PROGRAM Batch_Controller
  VAR_EXTERNAL
    Safety_OK : BOOL;
    Level : REAL;
    Temperature : REAL;
    Pressure : REAL;
    Weight : REAL;
    Ingredient_A_Request : BOOL;
    Ingredient_B_Request : BOOL;
    Discharge_Request : BOOL;
    Packaging_Request : BOOL;
    Mixer_Request : BOOL;
    Batch_State_Code : INT;
    Batch : ST_BATCH;
  END_VAR
  VAR
    Batch_Start : BOOL;
    Batch_Stop : BOOL;
    Batch_Reset : BOOL;
    Fill_A_Active : BOOL;
    Fill_A_Done : BOOL;
    Fill_B_Active : BOOL;
    Fill_B_Done : BOOL;
    Batch_Target : REAL;
    Mix_Active : BOOL;
    Mix_Done : BOOL;
    Mix_Timer : TON;
    Discharge_Active : BOOL;
    Discharge_Done : BOOL;
    Packaging_Active : BOOL;
    Packaging_Done : BOOL;
    Packaging_Timer : TON;
    Batch_Complete : BOOL;
    Batch_Start_Trig : R_TRIG;
  END_VAR
  VAR  (* added by the conversion: wires and edge detectors of the diagram *)
    _State_Transition12_ENO : BOOL;
    _State_Transition12_OUT : INT;
  END_VAR

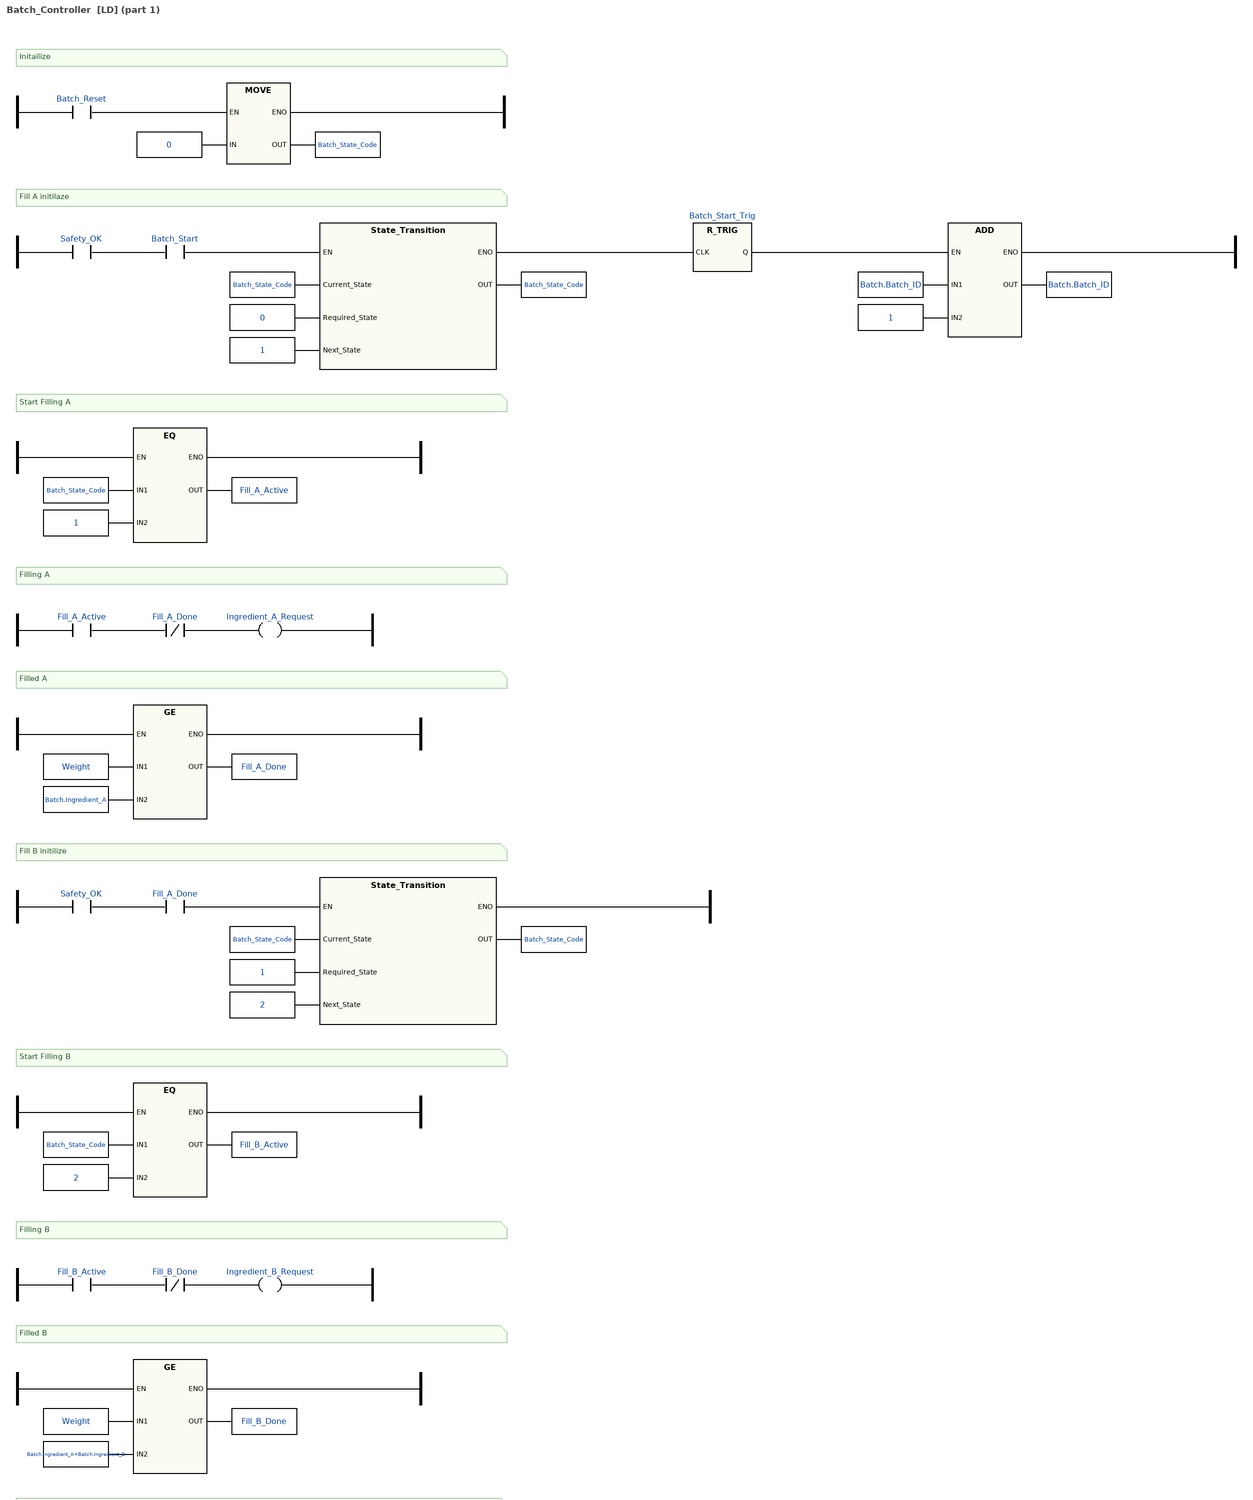
(* LD diagram, written out as Structured Text *)
(* Initailize *)
IF Batch_Reset THEN Batch_State_Code := 0; END_IF;
(* Fill A initilaze *)
_State_Transition12_OUT := State_Transition(EN := Safety_OK AND Batch_Start, Current_State := Batch_State_Code, Required_State := 0, Next_State := 1, ENO => _State_Transition12_ENO);
IF _State_Transition12_ENO THEN Batch_State_Code := _State_Transition12_OUT; END_IF;
Batch_Start_Trig(CLK := _State_Transition12_ENO);
IF Batch_Start_Trig.Q THEN Batch.Batch_ID := Batch.Batch_ID + 1; END_IF;
(* Start Filling A *)
Fill_A_Active := Batch_State_Code = 1;
(* Filling A *)
Ingredient_A_Request := Fill_A_Active AND NOT Fill_A_Done;
(* Filled A *)
Fill_A_Done := Weight >= Batch.Ingredient_A;
(* Fill B initilize *)
IF Safety_OK AND Fill_A_Done THEN Batch_State_Code := State_Transition(Batch_State_Code, 1, 2); END_IF;
(* Start Filling B *)
Fill_B_Active := Batch_State_Code = 2;
(* Filling B *)
Ingredient_B_Request := Fill_B_Active AND NOT Fill_B_Done;
(* Filled B *)
Fill_B_Done := Weight >= (Batch.Ingredient_A+Batch.Ingredient_B);
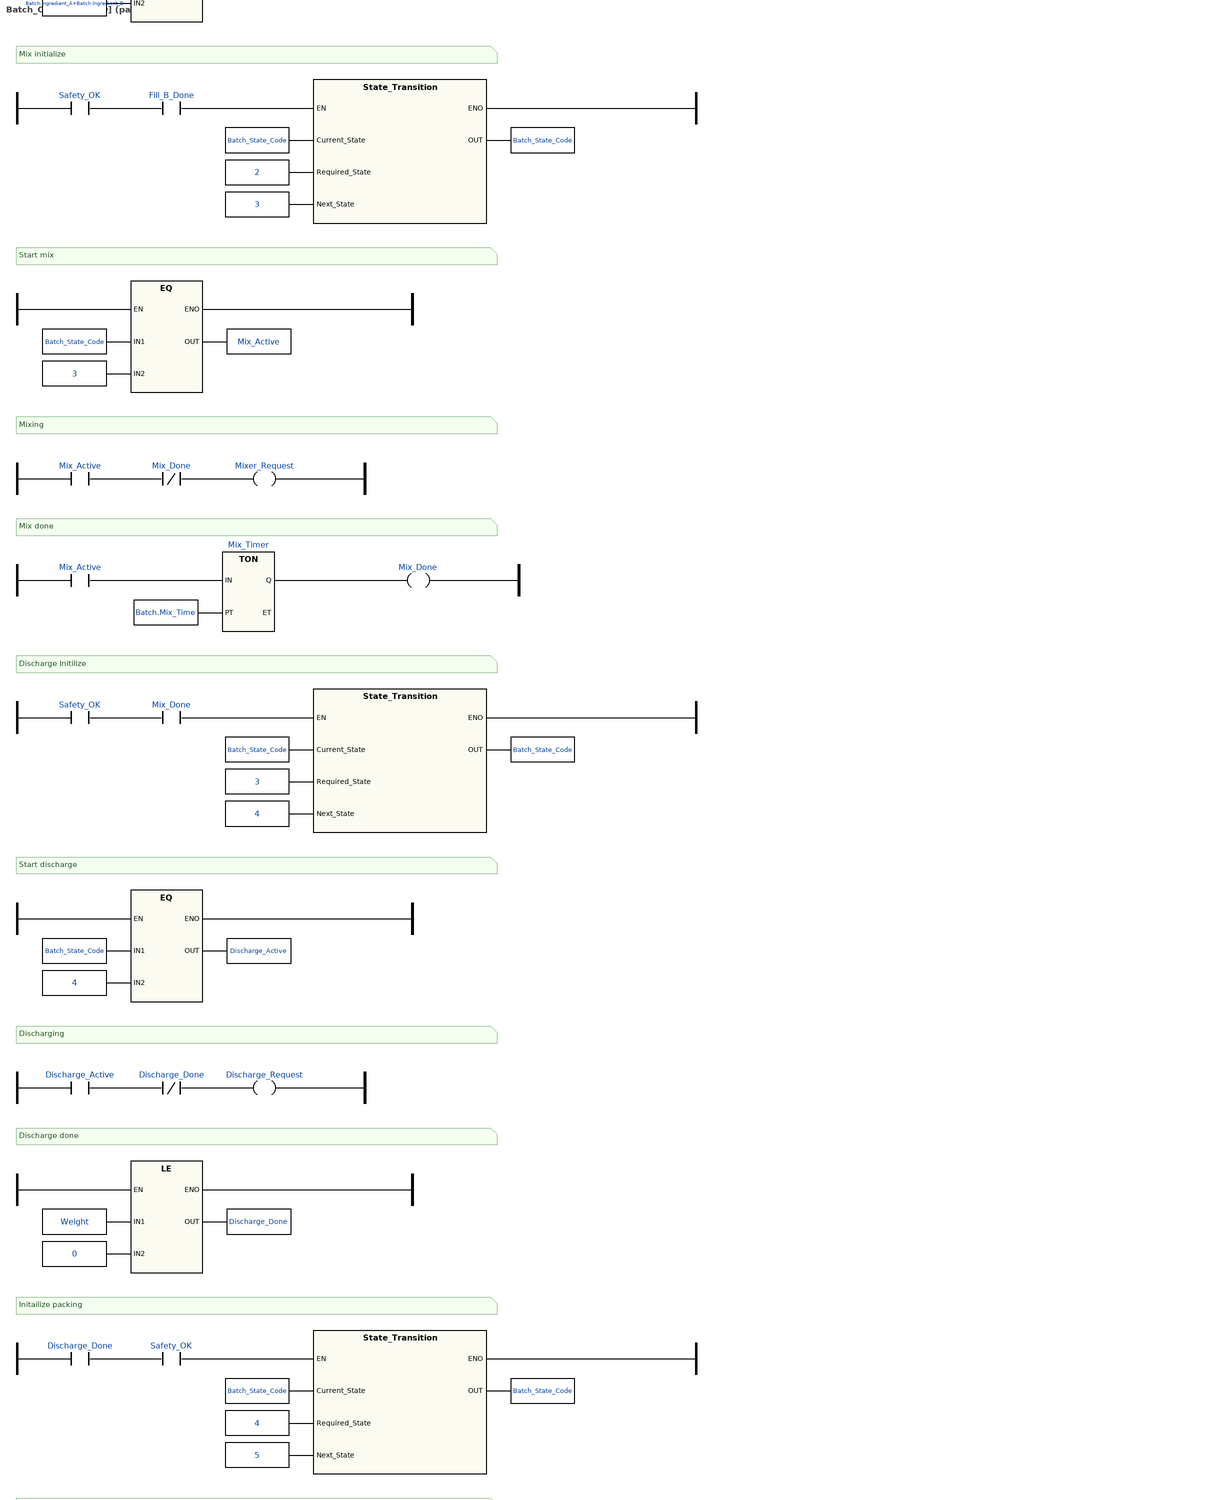
(* Mix initialize *)
IF Safety_OK AND Fill_B_Done THEN Batch_State_Code := State_Transition(Batch_State_Code, 2, 3); END_IF;
(* Start mix *)
Mix_Active := Batch_State_Code = 3;
(* Mixing *)
Mixer_Request := Mix_Active AND NOT Mix_Done;
(* Mix done *)
Mix_Timer(IN := Mix_Active, PT := Batch.Mix_Time);
Mix_Done := Mix_Timer.Q;
(* Discharge Initilize *)
IF Safety_OK AND Mix_Done THEN Batch_State_Code := State_Transition(Batch_State_Code, 3, 4); END_IF;
(* Start discharge *)
Discharge_Active := Batch_State_Code = 4;
(* Discharging *)
Discharge_Request := Discharge_Active AND NOT Discharge_Done;
(* Discharge done *)
Discharge_Done := Weight <= 0;
(* Initailize packing *)
IF Discharge_Done AND Safety_OK THEN Batch_State_Code := State_Transition(Batch_State_Code, 4, 5); END_IF;
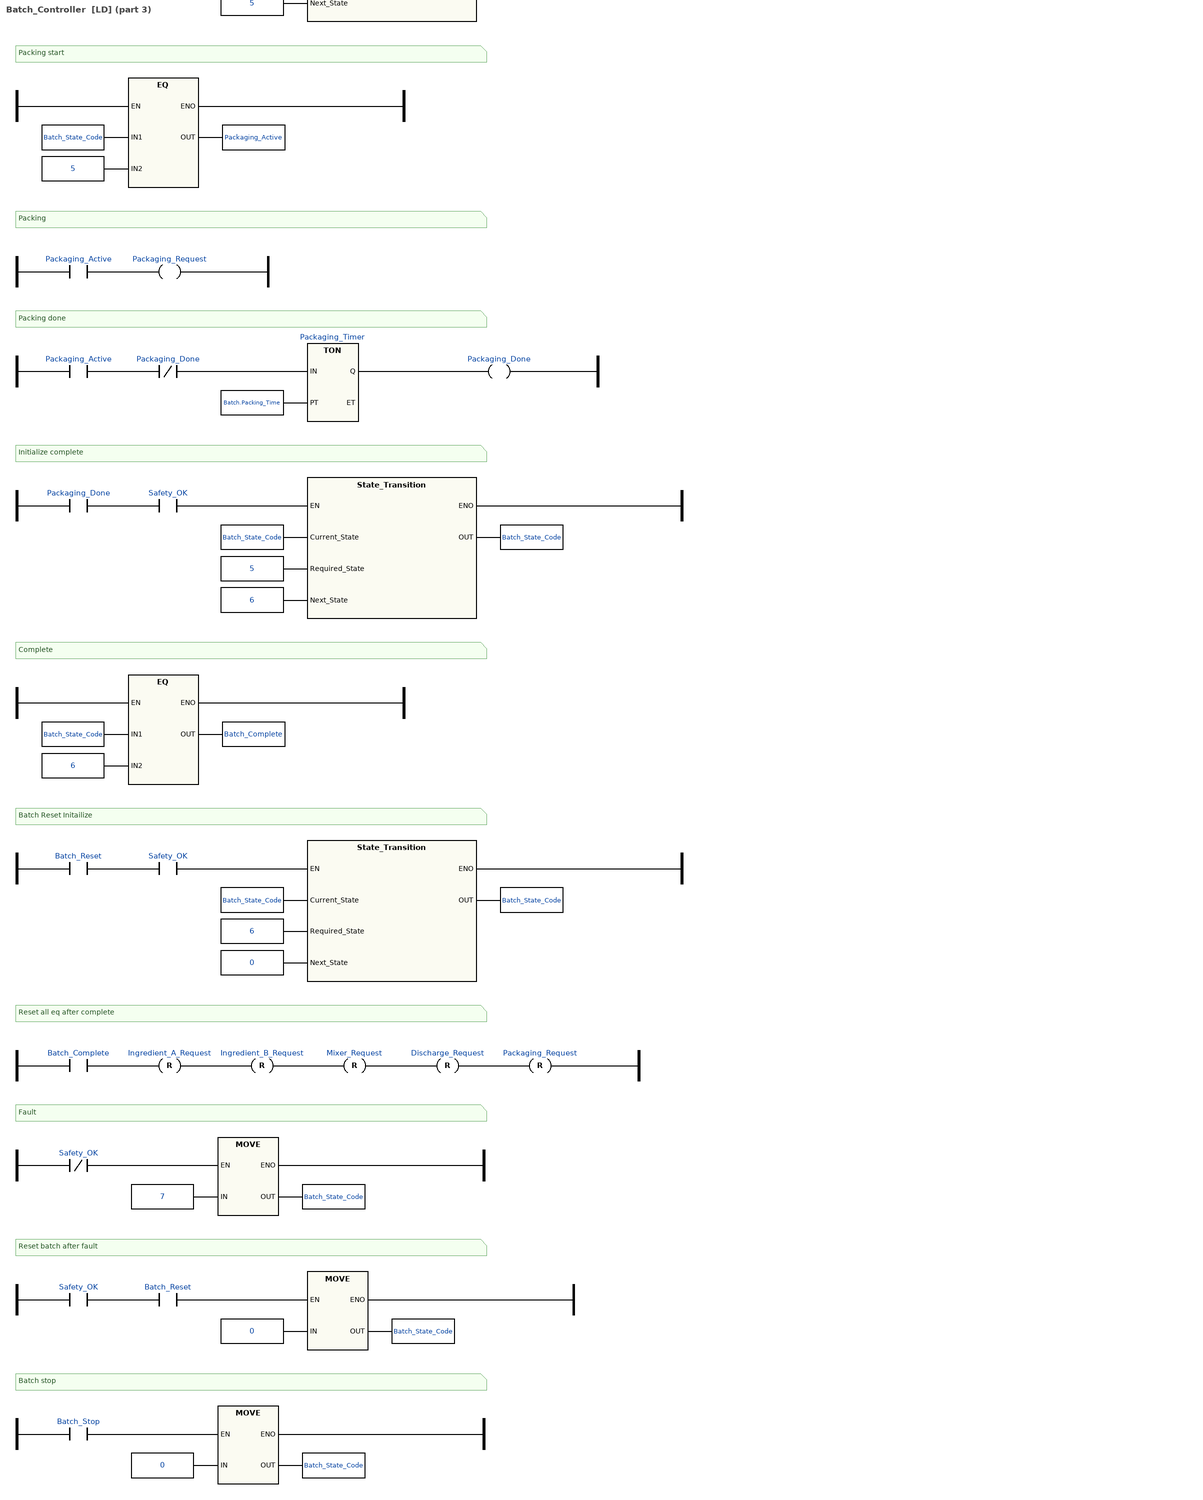
(* Packing start *)
Packaging_Active := Batch_State_Code = 5;
(* Packing *)
Packaging_Request := Packaging_Active;
(* Packing done *)
Packaging_Timer(IN := Packaging_Active AND NOT Packaging_Done, PT := Batch.Packing_Time);
Packaging_Done := Packaging_Timer.Q;
(* Initialize complete *)
IF Packaging_Done AND Safety_OK THEN Batch_State_Code := State_Transition(Batch_State_Code, 5, 6); END_IF;
(* Complete *)
Batch_Complete := Batch_State_Code = 6;
(* Batch Reset Initailize *)
IF Batch_Reset AND Safety_OK THEN Batch_State_Code := State_Transition(Batch_State_Code, 6, 0); END_IF;
(* Reset all eq after complete *)
IF Batch_Complete THEN Ingredient_A_Request := FALSE; END_IF;
IF Batch_Complete THEN Ingredient_B_Request := FALSE; END_IF;
IF Batch_Complete THEN Mixer_Request := FALSE; END_IF;
IF Batch_Complete THEN Discharge_Request := FALSE; END_IF;
IF Batch_Complete THEN Packaging_Request := FALSE; END_IF;
(* Fault *)
IF NOT Safety_OK THEN Batch_State_Code := 7; END_IF;
(* Reset batch after fault *)
IF Safety_OK AND Batch_Reset THEN Batch_State_Code := 0; END_IF;
(* Batch stop *)
IF Batch_Stop THEN Batch_State_Code := 0; END_IF;
END_PROGRAM
